FUNCTION_BLOCK FB_ControllerPalletStacker
VAR_INPUT
    CmdCollect     : BOOL;
    CmdEmpty       : BOOL;
    CmdReset       : BOOL;
    CmdStack       : BOOL;
    CmdStop        : BOOL;

    AutoMode       : BOOL;   // enables automatic sensor simulation
    AutoRun        : BOOL;   // starts repeated collecting cycles

    Door1Closed    : BOOL;
    Door2Closed    : BOOL;
    EStop        : BOOL;

    AutoDelayPalletBefore : TIME := T#2S;
    AutoDelayPalletInLift : TIME := T#2S;
    AutoDelayPinsOut      : TIME := T#1S;
    AutoDelayPinsIn       : TIME := T#1S;
    AutoCycleDelay        : TIME := T#2S;
END_VAR

VAR_IN_OUT
    Stacker           : FB_PalletStacker(DoorClosed:= Door1Closed); // change to your actual FB type
    PalletBeforeLift  : BOOL; // PalletBufferSensor.SensorWaarde1
    PalletInLift      : BOOL; // PalletInLiftSensor.SensorWaarde1
    PinsOutFb         : BOOL; // pins.PinsUit feedback (simulated)
    PinsInFb          : BOOL; // pins.PinsIn feedback (simulated)
END_VAR

VAR_OUTPUT
    SafetyPaused  : BOOL;
    AutoRunning   : BOOL;
    ActiveCmd     : INT;  // 0 none, 1 collect, 2 empty, 3 reset, 4 stack, 5 stop
END_VAR
	
	VAR
	AllDoorsClosed : BOOL;
	SafetyTrip      : BOOL;
	SafetyLatch     : BOOL;
	SafetyAck       : BOOL; // HMI button

    rCollect : R_TRIG;
    rEmpty   : R_TRIG;
    rReset   : R_TRIG;
    rStack   : R_TRIG;
    rStop    : R_TRIG;

    cmdLatched : INT;

    tPalletBefore : TON;
    tPalletIn     : TON;
    tPinsOut      : TON;
    tPinsIn       : TON;
    tAutoCycle    : TON;

    prevState : E_PalletStackerStatus;
END_VAR

// Safety
AllDoorsClosed := Door1Closed AND Door2Closed;
SafetyTrip := (NOT AllDoorsClosed) OR (EStop);

IF SafetyTrip THEN
    SafetyLatch := TRUE;
END_IF

IF SafetyAck AND NOT SafetyTrip THEN
    SafetyLatch := FALSE;
END_IF

SafetyPaused := SafetyTrip OR SafetyLatch;

// Pass combined safety into stacker
stacker(
    DoorClosed := AllDoorsClosed,
    EStopOk := NOT EStop,
    SafetyHold := SafetyLatch
);

IF SafetyPaused THEN
    Stacker.Stop();
    cmdLatched := 0;
    ActiveCmd := 0;
    AutoRunning := FALSE;
END_IF

// Edge detect commands
rCollect(CLK := CmdCollect);
rEmpty(CLK := CmdEmpty);

IF rCollect.Q THEN cmdLatched := 1; END_IF
IF rEmpty.Q THEN
    //Stacker.EmptyStack();
    //ActiveCmd := 2;
    cmdLatched := 0;
END_IF

// Looping collect mode
AutoRunning := AutoRun AND NOT SafetyPaused;

// Execute commands
IF NOT SafetyPaused THEN
    // Empty has priority and can interrupt Collect
    IF rEmpty.Q THEN
        Stacker.EmptyStack();
        ActiveCmd := 2;
        cmdLatched := 0;
    ELSIF ActiveCmd = 0 THEN
        IF cmdLatched <> 0 THEN
            CASE cmdLatched OF
                1: Stacker.CollectPallet();
                2: Stacker.EmptyStack();
            END_CASE
            ActiveCmd := cmdLatched;
            cmdLatched := 0;

        ELSIF AutoRunning AND (Stacker.State = E_PalletStackerStatus.Idle) THEN
            tAutoCycle(IN := TRUE, PT := AutoCycleDelay);
            IF tAutoCycle.Q THEN
                Stacker.CollectPallet();
                ActiveCmd := 1;
                tAutoCycle(IN := FALSE);
            END_IF
        ELSE
            tAutoCycle(IN := FALSE);
        END_IF
    ELSE
        IF Stacker.State = E_PalletStackerStatus.Idle THEN
            ActiveCmd := 0;
        END_IF
    END_IF
END_IF

END_FUNCTION_BLOCK

(* stored: Version 1.1.0.1
   POU FB_ControllerPalletStacker: Id {d94f743d-0e17-40db-8373-d42e5b0997e7}, SpecialFunc None *)
